TYPE T_PositiveDINT : DINT(0..2147483647); END_TYPE

(* stored: Version 1.1.0.1
   DUT T_PositiveDINT: Id {3c818d9c-2fd6-430b-988c-7ae45c148db1} *)
